PROGRAM MAIN_FBD
VAR
	rPosSenDis_mm : REAL;
	rPosSenDis_inch : REAL;
END_VAR

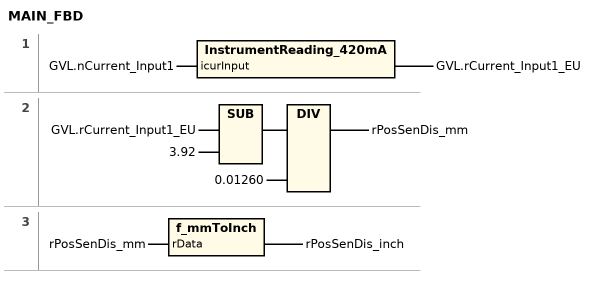
// NETWORK 1
GVL.rCurrent_Input1_EU := InstrumentReading_420mA(icurInput := GVL.nCurrent_Input1);

// NETWORK 2
rPosSenDis_mm := (GVL.rCurrent_Input1_EU - 3.92) / 0.01260;

// NETWORK 3
rPosSenDis_inch := f_mmToInch(rData := rPosSenDis_mm);

END_PROGRAM

(* stored: Version 1.1.0.1, ProductVersion 3.1.4024.12
   POU MAIN_FBD: Id {7005b1c0-7e07-4c3c-be1c-bb64bb3cb219}, SpecialFunc None *)
